TYPE ST_Feeder_HMI :
STRUCT
	bActivate		:BOOL;
	bDeactivate		:BOOL;
END_STRUCT
END_TYPE

(* stored: Version 1.1.0.1
   DUT ST_Feeder_HMI: Id {1c2e3f07-1986-49d5-8a4a-44dd92815213} *)
